{attribute 'OPC.UA.DA.JobMethod' := 'JobMethode_HorizontalMove'}
FUNCTION_BLOCK HRL_CB_AS_HorizontalMove
VAR
	AlwaysTrue : BOOL := TRUE;
	// Used for debugging purposes to display InputArguments of method call
	MethodCall_HorizontalMove : BOOL := FALSE; // used to store InputArg "MethodCall" from Start() method
	ResetMethodCall	: BOOL := FALSE;
	Direction : BOOL := FALSE; // defines movement direction
	callCounterStart : ULINT; // counts how many times the Start() method has been called
	callCounterCheckState : ULINT; // counts how many times the CheckState() method has been called
	callCounterAbort : ULINT; // counts how many times the Abort() method has been called
	
	// Variables to determine if a job has been started (Start() method has been called) or finished
	jobRunning : BOOL;
	jobFinished : BOOL;

	// State machine variable
	state : UDINT;
	
	// FB Intatziation Variable
	HRL_CB_HorizontalMove : AxisControl_MultipleInputSensors;
END_VAR
	
VAR_INPUT
	ESS: BOOL;
	LightBarrierSensor_01 : BOOL;
	LightBarrierSensor_02 : BOOL;
	AutomaticMode: BOOL;
END_VAR

VAR_OUTPUT
	Motor_Control : BOOL;
END_VAR

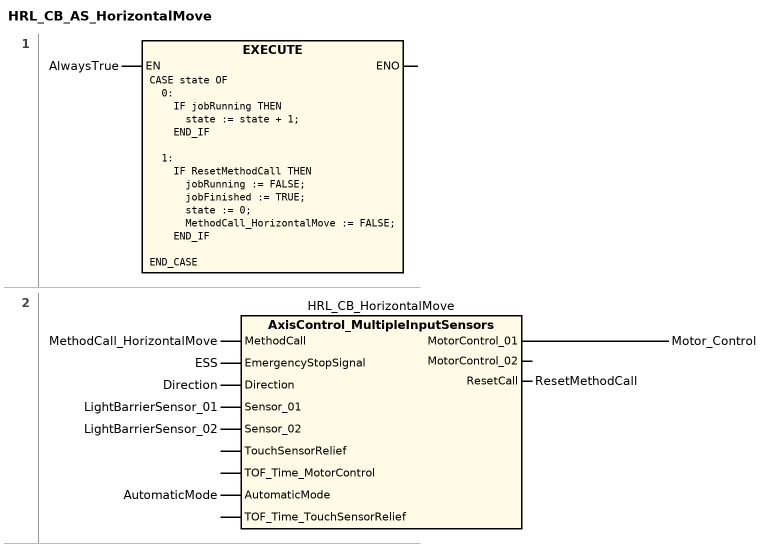
// NETWORK 1
IF AlwaysTrue THEN
    CASE state OF
    	0:
    		IF jobRunning THEN
    			state := state + 1;
    		END_IF
    		
    	1:
    		IF ResetMethodCall THEN
    			jobRunning := FALSE;
    			jobFinished := TRUE;
    			state := 0;
    			MethodCall_HorizontalMove := FALSE;
    		END_IF
    		
    END_CASE
END_IF

// NETWORK 2
HRL_CB_HorizontalMove(
    MethodCall := MethodCall_HorizontalMove,
    EmergencyStopSignal := ESS,
    Direction := Direction,
    Sensor_01 := LightBarrierSensor_01,
    Sensor_02 := LightBarrierSensor_02,
    AutomaticMode := AutomaticMode,
    ResetCall => ResetMethodCall); // AxisControl_MultipleInputSensors
Motor_Control := HRL_CB_HorizontalMove.MotorControl_01;

{attribute 'TcRpcEnable' := '1'}
METHOD Abort : HRESULT
VAR_INPUT
	hdl : UDINT; // Do not change, used by server.
END_VAR
callCounterAbort := callCounterAbort + 1;
END_METHOD

{attribute 'TcRpcEnable' := '1'}
METHOD CheckState : HRESULT
VAR_INPUT
	hdl : UDINT; // Do not change, used by server.
END_VAR
VAR_OUTPUT
	bBusy : BOOL; // Do not change. Used by server to find out if the job is finished
	
	// List of OutputArguments for OPC UA method, may be customized
	State : BOOL; // Abgeschlossener MethodCall
	MethodCall: BOOL; //Input Recall
END_VAR
callCounterCheckState := callCounterCheckState + 1;
IF NOT jobFinished THEN
	bBusy := TRUE; // job is not finished yet
	CheckState := 0; // no error
ELSE
	bBusy := FALSE; // job is finished
	CheckState := 0; // done, no error occured during execution (OPC UA StatusCode "GOOD")
	jobFinished := FALSE;
	State := ResetMethodCall;
	MethodCall := MethodCall_HorizontalMove;
END_IF
END_METHOD

{attribute 'TcRpcEnable' := '1'}
METHOD Start : HRESULT
VAR_INPUT
	// List of InputArguments for OPC UA method, may be customized
	MethodCall : BOOL; // some description
	MovementDirection : BOOL;	
END_VAR
VAR_OUTPUT
	hdl : UDINT; // Do not change, used by server.
END_VAR
callCounterStart := callCounterStart + 1;

MethodCall_HorizontalMove := MethodCall;
MovementDirection := Direction;

jobRunning := TRUE;
Start := 0; // no error occured, e.g. while parsing the input arguments (0 = OPC UA StatusCode "GOOD")
END_METHOD

END_FUNCTION_BLOCK

(* stored: Version 1.1.0.1, ProductVersion 3.1.4024.15
   POU HRL_CB_AS_HorizontalMove: Id {e5740522-dfa1-4a36-b236-0740e0d326ba}, SpecialFunc None
   Method Abort: Id {f5647571-a28f-4042-beec-29e749c636d5}
   Method CheckState: Id {060c9808-54d1-4d1e-ab68-457cc9b822f4}
   Method Start: Id {5edcf620-8359-429a-9afe-262ce45d41b7} *)
